TYPE "TAx_Speed_Sts"
VERSION : 0.1
// Block: TAx_Speed_Sts
   STRUCT
      AlarmPresence : Bool;
      WarningPresence : Bool;
      Enabled : Bool;
      Done : Bool;
      Standstill : Bool;
      RstHWDone : Bool;
      AtProgrammedSpeed : Bool;
      MoveMinusPermitted : Bool;
      MovePlusPermitted : Bool;
      ActualSpeed : LReal;
   END_STRUCT;

END_TYPE
